TYPE (* A service representation for the Arrowhead framework 4.0 *)
  (* Standard: 61499-2 *)
  (* Version 1.0, 2018-09-26, Jose Cabral, fortiss GmbH *)
  (* ASN.1 tag APPLICATION 1 *)
  ArrowheadService : STRUCT
    systemName : WSTRING; (* Identification of the system *)
    address : WSTRING; (* Address of the offered services *)
    port : DINT; (* Port of the of the offered services *)
    authenticationInfo : WSTRING; (* Authentication info of the system *)
  END_STRUCT;
END_TYPE
